FUNCTION_BLOCK ValueSum EXTENDS AbstractApplier
VAR
	valueObject :IHaveValue;
	mySum :LREAL;
END_VAR

(*

short summary
=================
Methode to accept an object.
Example:
NumberIncrementer.accept(Number);

.. <legal notes>

legal notes
=================
| SPDX-FileCopyrightText: © 2022 ekvip automation GmbH <info@ekvip.de>
| SPDX-License-Identifier: Apache-2.0
| For details check: Apache-2.0_

.. _Apache-2.0: https://www.apache.org/licenses/LICENSE-2.0

.. </legal notes>

parameters
=========================

*)
METHOD accept : CNM_CollectionInterfaces.CNM_ReturnTypes.SingleExecutionResult
VAR_INPUT
	(*object to accept*)
	object	: CNM_CollectionInterfaces.CNM_AbstractObject.IObject;
END_VAR
IF(__QUERYINTERFACE(object, THIS^.valueObject))THEN
	accept := CNM_ReturnTypes.SingleExecutionResult.SUCCESS;
ELSE
	accept := CNM_ReturnTypes.SingleExecutionResult.ERROR;
END_IF
END_METHOD

(*

short summary
=================
A method to apply the concrete action on the given object (THIS^.object)

.. <legal notes>

legal notes
=================
| SPDX-FileCopyrightText: © 2022 ekvip automation GmbH <info@ekvip.de>
| SPDX-License-Identifier: Apache-2.0
| For details check: Apache-2.0_

.. _Apache-2.0: https://www.apache.org/licenses/LICENSE-2.0

.. </legal notes>

parameters
=========================
:return: CNM_ReturnTypes.ExecutionState

*)
METHOD apply : CNM_CollectionInterfaces.CNM_ReturnTypes.SingleExecutionState
VAR_INPUT
	(*control bit to start or abort the application, should to be active until the ExecutionState is SUCCESS*)
	execute	: BOOL;
END_VAR
RETURN (NOT execute);

apply := CNM_ReturnTypes.SingleExecutionState.ERROR;

RETURN (THIS^.isObjectNull(THIS^.valueObject));

apply := CNM_ReturnTypes.SingleExecutionState.SUCCESS;
THIS^.sum := THIS^.sum + THIS^.valueObject.value;
END_METHOD

(*

short summary
=================
This abstract property returns the class name of the concrete object, 
which is useful for logging/debugging purpose or to check the class name
for ``__DELETE`` in factories (sometimes it's necessary to do more 
than just to free the memory).

.. <legal notes>

legal notes
=================
| SPDX-FileCopyrightText: © 2022 ekvip automation GmbH <info@ekvip.de>
| SPDX-License-Identifier: Apache-2.0
| For details check: Apache-2.0_

.. _Apache-2.0: https://www.apache.org/licenses/LICENSE-2.0

.. </legal notes>

*)
PROPERTY className : CNM_AbstractObject.ClassName
GET
className := 'AOC.ValueSum';
END_GET
END_PROPERTY

PROPERTY sum : LREAL
GET
sum := THIS^.mySum;
END_GET
SET
THIS^.mySum := sum;
END_SET
END_PROPERTY

END_FUNCTION_BLOCK

(* stored: Version 1.1.0.1
   POU ValueSum: Id {3ec42af7-f5d5-4ca1-a3db-3ddee1c8dc28}, SpecialFunc None
   Method accept: Id {0751e69f-a6a2-4b2f-a8b6-e674aab29d11}
   Method apply: Id {4bfc40b2-2e65-4325-a442-04dfeada8c78}
   Property className: Id {3a7d4571-9147-44f0-bef9-d32ffcb20ebd}
   Get Get: Id {771953c3-e3fa-490b-a5a5-08404ff7d78a}
   Property sum: Id {f63c941b-c6a9-4e27-8b47-e115b7bda489}
   Get Get: Id {32ffe4ab-d42c-4f8a-b732-0ee335b0e25f}
   Set Set: Id {659b2951-73b8-420c-b34f-d84ac9512ea0} *)
